// TIA Portal V20 export
TYPE "UDT_Interlock_TE_FSS"
   STRUCT
      S1_Arrival : Bool;   // MESA DE CARGA E1
      S1_Rotative : Bool;   // MESA DE CARGA E1
      S1_Complete : Bool;   // MESA DE CARGA E1
      MA_PickUpOK_S1 : Bool;   // MESA DE CARGA E1
      S3_Arrival : Bool;   // MESA DE CARGA E3
      S3_Rotative : Bool;   // MESA DE CARGA E3
      S3_Complete : Bool;   // MESA DE CARGA E3
      MA_PickUpOK_S3 : Bool;   // MESA DE CARGA E3
      TE_OFFLine_carga : Bool;   // OFF Line del TE
      TE_PotenciaOK_carga : Bool;   // Potencia OK del TE
      Byte1_bit2 : Bool;
      Byte1_bit3 : Bool;
      Byte1_bit4 : Bool;
      Byte1_bit5 : Bool;
      Byte1_bit6 : Bool;
      Byte1_bit7 : Bool;
      E1_Arrival : Bool;   // MESA DE DESCARGA S1
      E1_Rotative : Bool;   // MESA DE DESCARGA S1
      MA_DepositOK_E1 : Bool;   // MESA DE DESCARGA S1
      MA_Complete_E1 : Bool;   // MESA DE DESCARGA S1
      E3_Arrival : Bool;   // MESA DE DESCARGA S3
      E3_Rotative : Bool;   // MESA DE DESCARGA S3
      MA_Complete_E4 : Bool;   // MESA DE DESCARGA S3
      MA_DepositOK_E3 : Bool;   // MESA DE DESCARGA S3
      MA_Complete_E3 : Bool;   // MESA DE DESCARGA S3
      TE_OFFLine_descarga : Bool;   // OFF Line del TE
      TE_PotenciaOK_descarga : Bool;   // Potencia OK del TE
      Byte3_bit3 : Bool;
      Byte3_bit4 : Bool;
      Byte3_bit5 : Bool;
      Byte3_bit6 : Bool;
      Byte3_bit7 : Bool;
   END_STRUCT;
END_TYPE
